FUNCTION_BLOCK FB_Predictive
VAR PERSISTENT
	rStatCoefMin:REAL:=0.0025;
	rFreqMean:REAL:=1.5;
	rFreqDev:REAL:=1.5;
END_VAR
VAR_INPUT
	bReset:BOOL;
END_VAR
VAR_OUTPUT
	bWarningMean:BOOL;
	bWarningDev:BOOL;
END_VAR
VAR
	fbStatistic:FB_Statistic;
	fbStatisticDev:FB_Statistic;
END_VAR

METHOD PRIVATE M_check
VAR_INPUT
END_VAR
IF THIS^.fbStatistic.bSaved THEN
	THIS^.bWarningMean	:= 	THIS^.fbStatistic.M_is_typical(freqTypical:=THIS^.rFreqMean);
	THIS^.bWarningDev 	:= 	THIS^.fbStatisticDev.M_is_typical(freqTypical:=THIS^.rFreqDev);
ELSE
	THIS^.bWarningMean:=FALSE;
	THIS^.bWarningDev:=FALSE;
END_IF
END_METHOD

METHOD M_run
VAR_INPUT
	rValue:REAL;
END_VAR
IF THIS^.bReset THEN
	THIS^.fbStatistic.bReset:=TRUE;
	THIS^.fbStatisticDev.bReset:=TRUE;
	THIS^.bReset:=FALSE;
END_IF

THIS^.fbStatistic.M_run(rStatCoefMin:=THIS^.rStatCoefMin,
						rCurrentValue:=rValue);
						
THIS^.fbStatisticDev.M_run(	rStatCoefMin:=THIS^.rStatCoefMin,
							rCurrentValue:=THIS^.fbStatistic.Data.rDev);
							
THIS^.M_check();
END_METHOD

END_FUNCTION_BLOCK

(* stored: Version 1.1.0.1, ProductVersion 3.1.4024.15
   POU FB_Predictive: Id {2036f947-9e4d-47ed-8629-ab9129c21978}, SpecialFunc None
   Method M_check: Id {74b4c88d-131c-4819-b217-dc360cc3402f}
   Method M_run: Id {6069251c-0dd0-4f1f-812e-75f9ff48d900} *)
